//<DataManagerDeclarations>
// Function block for data maipulation must extend from TcoData.TcoDataExchange.
FUNCTION_BLOCK TcoDataManager EXTENDS TcoData.TcoDataExchange
VAR
	// This is the structure that contains the actual data we will work with. The `STRUCT` must extend `TcoData.TcoEntity`
    _data : SandboxData;
END_VAR
//</DataManagerDeclarations>

//----------------------------------
//<DataManagerSuperCall>

// IMPLEMENTATION BODY OF FUNCTION BLOCK

// IMPORTANT: SUPER CALL HERE IS REQUIRED TO CALL THE DATA MANAGER TASKS!!!
SUPER^();

//</DataManagerSuperCall>
//----------------------------------

PROPERTY Data : REFERENCE TO SandboxData
GET
Data REF= _data;
END_GET
END_PROPERTY

END_FUNCTION_BLOCK

(* stored: Version 1.1.0.1, ProductVersion 3.1.4024.9
   POU TcoDataManager: Id {cbedc24e-3653-0ddc-2b27-80848f6cc570}, SpecialFunc None
   Property Data: Id {2597f0fe-0638-0425-240d-70cbc2d30219}
   Get Get: Id {574052f0-d5c9-0f6e-2355-c06a1e3971c5} *)
